# EPICS substitutions: mc11/tpmacApp/Db/autohome.substitutions
file "db/autohome.db"
{
pattern
{SYS,                  DEV,                 PLC,  PORT  }
{"XF:16IDC-ES:InAir",  "{Slt:G2-Ax:X}",     8,    P0    }
{"XF:16IDC-ES:InAir",  "{Slt:G2-Ax:dX}",    9,    P0    }
{"XF:16IDC-ES:InAir",  "{Slt:G2-Ax:Y}",     10,   P0    }
{"XF:16IDC-ES:InAir",  "{Slt:G2-Ax:dY}",    11,   P0    }
{"XF:16IDC-ES",        "{BS:SAXS-Ax:X}",    12,   P0    }
{"XF:16IDC-ES",        "{BS:SAXS-Ax:Y}",    13,   P0    }
}
